Staubli VAL3: getSession.pgx

public program getSession(string& x_sName[] (dimensions=1))
  local num l_nPos[2]
  local num l_nSize
begin
  l_nPos=find(sPathTraj,"Disk://session")
  if l_nPos==-1
    // give back the session name
    x_sName=""
  else
    l_nPos[1]=find(sPathTraj,"/saveTraj/")
    l_nSize=l_nPos[1]-l_nPos-len("Disk://session/")
    x_sName=mid(sPathTraj,l_nSize,l_nPos+len("Disk://session/"))
  endIf
end
